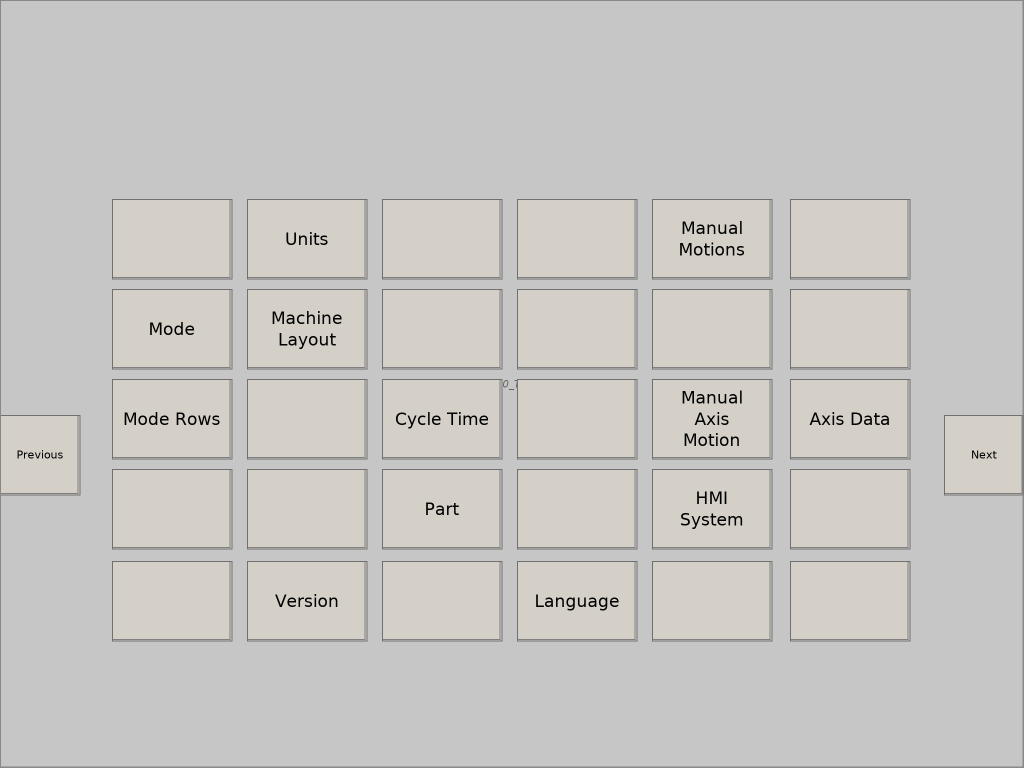
VISUALIZATION Men_030_MenuScreen  // 1024x768
    Frame (0,0 1024x768)
        shows Tmp_000_Template(header := gHMIData.hmiHeader)
    Button (112,199 120x80), text list: ''
        OnMouseDown: execute { gHMIButtons.gAnyButtonPressed := TRUE; }
    Button (247,199 120x80), "Units", text list: ''
        OnMouseDown: execute { gHMIButtons.gAnyButtonPressed := TRUE; }
        OnMouseDown: change screen: Unt_401_Units
    Button (382,199 120x80), text list: ''
        OnMouseDown: execute { gHMIButtons.gAnyButtonPressed := TRUE; }
    Button (517,199 120x80), text list: ''
        OnMouseDown: execute { gHMIButtons.gAnyButtonPressed := TRUE; }
    Button (652,199 120x80), "Manual Motions", text list: ''
        OnMouseClick: change screen: Mot_010_Motions
        OnMouseDown: execute { gHMIButtons.gAnyButtonPressed := TRUE; }
    Button (790,199 120x80), text list: ''
        OnMouseDown: execute { gHMIButtons.gAnyButtonPressed := TRUE; }
    Button (112,289 120x80), "Mode", text list: ''
        OnMouseDown: execute { gHMIButtons.gAnyButtonPressed := TRUE; }
        OnMouseDown: change screen: Mod_001_ModeScreen
    Button (247,289 120x80), "Machine Layout", text list: ''
        OnMouseDown: execute { gHMIButtons.gAnyButtonPressed := TRUE; }
        OnMouseDown: change screen: Lay_040_MachineLayout
    Button (382,289 120x80), text list: ''
        OnMouseDown: execute { gHMIButtons.gAnyButtonPressed := TRUE; }
    Button (517,289 120x80), text list: ''
        OnMouseDown: execute { gHMIButtons.gAnyButtonPressed := TRUE; }
    Button (652,289 120x80), text list: ''
        OnMouseDown: execute { gHMIButtons.gAnyButtonPressed := TRUE; }
    Button (790,289 120x80), text list: ''
        OnMouseDown: execute { gHMIButtons.gAnyButtonPressed := TRUE; }
    Button (112,379 120x80), "Mode Rows", text list: ''
        OnMouseDown: execute { gHMIButtons.gAnyButtonPressed := TRUE; }
        OnMouseDown: change screen: Mod_002_ModeScreenRows
    Button (247,379 120x80), text list: ''
        OnMouseDown: execute { gHMIButtons.gAnyButtonPressed := TRUE; }
    Button (382,379 120x80), "Cycle Time", text list: ''
        OnMouseDown: execute { gHMIButtons.gAnyButtonPressed := TRUE; }
        OnMouseDown: change screen: Prc_501_Cycle
    Button (517,379 120x80), text list: ''
        OnMouseDown: execute { gHMIButtons.gAnyButtonPressed := TRUE; }
    Button (652,379 120x80), "Manual Axis Motion", text list: ''
        OnMouseDown: execute { gHMIButtons.gAnyButtonPressed := TRUE; }
        OnMouseDown: change screen: Mot_011_Axis
    Button (790,379 120x80), "Axis Data", text list: ''
        OnMouseDown: execute { gHMIButtons.gAnyButtonPressed := TRUE; }
        OnMouseDown: change screen: Unt_402_Axis
    Button (112,469 120x80), text list: ''
        OnMouseDown: execute { gHMIButtons.gAnyButtonPressed := TRUE; }
    Button (247,469 120x80), text list: ''
        OnMouseDown: execute { gHMIButtons.gAnyButtonPressed := TRUE; }
    Button (382,469 120x80), "Part", text list: ''
        OnMouseDown: execute { gHMIButtons.gAnyButtonPressed := TRUE; }
        OnMouseDown: change screen: Prc_500_Part
    Button (517,469 120x80), text list: ''
        OnMouseDown: execute { gHMIButtons.gAnyButtonPressed := TRUE; }
    Button (652,469 120x80), "HMI System", text list: ''
        OnMouseDown: execute { gHMIButtons.gAnyButtonPressed := TRUE; }
        OnMouseDown: change screen: Sys_901_HMISystem
    Button (790,469 120x80), text list: ''
        OnMouseDown: execute { gHMIButtons.gAnyButtonPressed := TRUE; }
    Button (112,561 120x80), text list: ''
        OnMouseDown: execute { gHMIButtons.gAnyButtonPressed := TRUE; }
    Button (247,561 120x80), "Version", text list: ''
        OnMouseDown: execute { gHMIButtons.gAnyButtonPressed := TRUE; }
        OnMouseDown: change screen: Sys_902_Version
    Button (382,561 120x80), text list: ''
        OnMouseDown: execute { gHMIButtons.gAnyButtonPressed := TRUE; }
    Button (517,561 120x80), "Language", text list: ''
        OnMouseDown: execute { gHMIButtons.gAnyButtonPressed := TRUE; }
        OnMouseDown: change screen: Unt_403_Language
    Button (652,561 120x80), text list: ''
        OnMouseDown: execute { gHMIButtons.gAnyButtonPressed := TRUE; }
    Button (790,561 120x80), text list: ''
        OnMouseDown: execute { gHMIButtons.gAnyButtonPressed := TRUE; }
    Group (0,415 1024x80)
        Button (0,0 80x80), "Previous"
            OnMouseClick: change screen: Men_032_MenuScreen_3
            OnMouseDown: execute { gHMIButtons.gAnyButtonPressed := TRUE; }
        Button (944,0 80x80), "Next"
            OnMouseClick: change screen: Men_031_MenuScreen_2
            OnMouseDown: execute { gHMIButtons.gAnyButtonPressed := TRUE; }
END_VISUALIZATION

(* stored: Version 1.1.0.1, ProductVersion 3.1.4024.11
   Visu Men_030_MenuScreen: Id {fcfc6bab-7c77-4a3a-b5c7-4b3a5f95aa3a} *)
